(* CODESYS project e!C_CanLayer2_Test_1.ecp

Project tree, tasks and I/O mapping:
  Controller : 750-8206 PFC200 2ETH RS CAN DPS, WAGO, order no. 0750-8206, version 5.11.1.16
    application Application
      task PLC_Task (cyclic, interval t#10ms, priority 14) calls PLC_PRG
      program PLC_PRG [CFC]
      data type typCanLayer2RxSchedule
      data type typCanLayer2TxSchedule
      global variables GVL_Constants
      program CAN_Layer2_Driver [ST]: CanLayer2RxScheduler, CanLayer2TxScheduler
      global variables GVL_Variables
      data type typCanMsg
    DeviceAdapter
    Kbus : Kbus, WAGO, version 1.4.0.2
        unmapped channels: K-BUS diagnostics
      _8_DO_DI_Generic : 075x-8DO8DI, WAGO, order no. 075x-8DO8DI, version 0.0.0.13
          settings: K-BUS Module slot index = 1
          unmapped channels: _IN, _OUT
        DeviceAdapter
      RS_232_RS_485_Interface_adjustable : 0750-0652, WAGO, order no. 0750-0652, version 0.0.0.25
          settings: K-BUS Module slot index = 2
          unmapped channels: _INPUTCHANNEL, _OUTPUTCHANNEL
        DeviceAdapter
    MODBUS
      MODBUS : MODBUS, WAGO, order no. n/a, version 1.1.1.15
    PROFIBUS
      PROFIBUS : PROFIBUS, WAGO, version 1.0.0.0 (disabled)
    CANbus
      WAGO_CAN_LAYER2_DEVICE : WAGO CAN Layer2 Device, WAGO, version 3.5.4.9
    Serial
      COM1 : COM1, WAGO, version 0.0.0.19
*)

// Controller/Application/typCanLayer2RxSchedule
TYPE typCanLayer2RxSchedule :
STRUCT
	udiTimeout: UDINT := 0;
	dwId: DWORD := 16#0000_0701;(* Set MSB = TRUE if 29bit ID:  dwId = 16#8xxx_xxxx *)
	diPktCnt: DINT;
	diPktCnt_old: DINT;
	diPktDeltaCnt: DINT;
	diRegisterIdResult: CANCFG.eCanFnReturn := CanNoIdx;
	udiPktDeltaTime: UDINT; (* Delta time between each packet in one channel, in msec *)
	udiPktArrivalTime: UDINT; (* Arrival time between each packet in one channel, in msec *)
	udiPktArrivalTime_old: UDINT; (* Last arrival time between each packet in one channel, in msec *)
	TON_CanRxMonitor: TON;
	tCanRxMonitorTimeout: TIME := T#5S;
	tCanRxMonitorElapsed: TIME;
	xCanRxMonitorAlarm: BOOL;
	atypMsgFifo: ARRAY[1..GVL_Constants.LIM_OF_CANJ1939_MSG_FIFO] OF typCanMsg;
	abMsg: ARRAY [1..8] OF BYTE;
END_STRUCT
END_TYPE

// Controller/Application/typCanLayer2TxSchedule
TYPE typCanLayer2TxSchedule :
STRUCT
	TON_TxErrorMonitor : TON;
	TON_TxCyclicMonitor : TON;
	TON_TxGapMonitor : TON;
	tTxError : TIME := T#5000MS;
	tTxInterval : TIME := T#200MS;
	tTxMinGap : TIME := T#100MS;
	udiTimeout: UDINT := 0;
	bScheduleType: BYTE := 1; (* 1 = cyclic,  2 = event *)
	xTxEvent: BOOL; (* send trigger,  only valid if bScheduleType = 2 *)
	dwId: DWORD := 16#0000_0240;(* Set MSB = TRUE if 29bit ID:  dwId = 16#8xxx_xxxx *)
	dwDlc: DWORD := 3;
	diPktCnt: DINT;
	diSendResult: DINT;
	diRegisterIdResult: CANCFG.eCanFnReturn;
	abMsg: ARRAY [1..8] OF BYTE := [16#AA, 16#AA, 16#AA];
END_STRUCT
END_TYPE

// Controller/Application/typCanMsg
TYPE typCanMsg :
STRUCT
	abMsg: ARRAY [1..8] OF BYTE;
END_STRUCT
END_TYPE

// Controller/Application/GVL_Constants
VAR_GLOBAL CONSTANT
	LIM_OF_CAN_LAYER2_TX_CHANNELS: INT := 3;
	LIM_OF_CAN_LAYER2_RX_CHANNELS: INT := 3;
	LIM_OF_CANJ1939_MSG_FIFO: INT := 20;
END_VAR

// Controller/Application/GVL_Variables
VAR_GLOBAL

	bEngine_A_State: BYTE;
	bEngine_A_Ctrl: BYTE;

	TON_CanRxMonitor: TON;
	tCanRxMonitorTimeout: TIME := T#5S;
	tCanRxMonitorElapsed: TIME;
	xCanRxMonitorAlarm: BOOL;
	
	atypCanLayer2RxSchedule : ARRAY[1..LIM_OF_CAN_LAYER2_RX_CHANNELS] OF typCanLayer2RxSchedule :=
		[
			(
				udiTimeout := 0,
				dwId := 16#0000_0701,
				diRegisterIdResult := CanNoIdx
			),
			(
				udiTimeout := 0,
				dwId := 16#0000_0181,
				diRegisterIdResult := CanNoIdx
			),
			(
				udiTimeout := 0,
				dwId := 16#8CF0_0300(* MSB: activates 29bit ID *),
				diRegisterIdResult := CanNoIdx
			)
		];

	atypCanLayer2TxSchedule : ARRAY[1..LIM_OF_CAN_LAYER2_TX_CHANNELS] OF typCanLayer2TxSchedule :=
		[
			(
				bScheduleType := 1,
				udiTimeout := 0,
				tTxInterval := T#500MS,
				tTxMinGap := T#100MS,
				dwId := 16#0000_0240,
				dwDlc := 3,
				abMsg := [16#AA, 16#AA, 16#AA]
			),
			(
				bScheduleType := 1,
				udiTimeout := 0,
				tTxInterval := T#500MS,
				tTxMinGap := T#100MS,
				dwId := 16#0000_0202,
				dwDlc := 3,
				abMsg := [16#BB, 16#BB, 16#BB]
			),
			(
				bScheduleType := 1,
				udiTimeout := 0,
				tTxInterval := T#500MS,
				tTxMinGap := T#100MS,
				dwId := 16#8CD0_0300(* MSB: activates 29bit ID *),
				dwDlc := 3,
				abMsg := [16#CC, 16#CC, 16#CC]
			)
		];

END_VAR

// Controller/Application/PLC_PRG
PROGRAM PLC_PRG
VAR


END_VAR

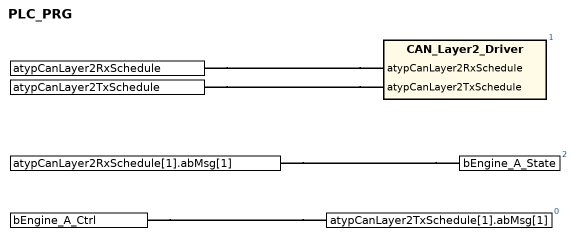
atypCanLayer2TxSchedule[1].abMsg[1] := bEngine_A_Ctrl;
CAN_Layer2_Driver(atypCanLayer2RxSchedule := atypCanLayer2RxSchedule, atypCanLayer2TxSchedule := atypCanLayer2TxSchedule);
bEngine_A_State := atypCanLayer2RxSchedule[1].abMsg[1];

END_PROGRAM

// Controller/Application/CAN_Layer2_Driver
PROGRAM CAN_Layer2_Driver
VAR_IN_OUT
	atypCanLayer2RxSchedule : ARRAY[1..LIM_OF_CAN_LAYER2_RX_CHANNELS] OF typCanLayer2RxSchedule;
	atypCanLayer2TxSchedule : ARRAY[1..LIM_OF_CAN_LAYER2_TX_CHANNELS] OF typCanLayer2TxSchedule;
END_VAR
VAR
	iCanLayer2RxChanIndex: INT;
	iCanLayer2TxChanIndex: INT;
	iCanRxPktIndex: INT;
	iCanRxPktIndexLim: INT;
	eCanL2ErrorCode: DINT;
	abMsg: ARRAY[1..8] OF BYTE;
END_VAR




CanLayer2RxScheduler();

CanLayer2TxScheduler();

ACTION CanLayer2RxScheduler:

(* Get Rx Packets *)
FOR iCanLayer2RxChanIndex := 1 TO LIM_OF_CAN_LAYER2_RX_CHANNELS DO
	IF (atypCanLayer2RxSchedule[iCanLayer2RxChanIndex].diRegisterIdResult <> CanFnOk) THEN
		(* IF CAN port is used for CAN Layer 2 and CANopen Master: *)
		(*atypCanLayer2RxSchedule[iCanLayer2RxChanIndex].diRegisterIdResult := WAGO_CANopen_Manager.RegisterId(eRegFlag := canRegisterId, dwId := atypCanLayer2RxSchedule[iCanLayer2RxChanIndex].dwId);*)

		(* IF CAN port is used for CAN Layer 2 and CANopen Slave: *)
		(*atypCanLayer2RxSchedule[iCanLayer2RxChanIndex].diRegisterIdResult := WAGO_CANopen_Local_Device.RegisterId(eRegFlag := canRegisterId, dwId := atypCanLayer2RxSchedule[iCanLayer2RxChanIndex].dwId);*)

		(* IF CAN port is used for CAN Layer 2 only: *)
		atypCanLayer2RxSchedule[iCanLayer2RxChanIndex].diRegisterIdResult := WAGO_CAN_LAYER2_Device.RegisterId(eRegFlag := canRegisterId, dwId := atypCanLayer2RxSchedule[iCanLayer2RxChanIndex].dwId);
	END_IF
	IF (atypCanLayer2RxSchedule[iCanLayer2RxChanIndex].diRegisterIdResult = CanFnOk) THEN
		GVL_Variables.TON_CanRxMonitor(IN:= TRUE, PT := GVL_Variables.tCanRxMonitorTimeout, ET=> GVL_Variables.tCanRxMonitorElapsed, Q=> GVL_Variables.xCanRxMonitorAlarm);
		atypCanLayer2RxSchedule[iCanLayer2RxChanIndex].TON_CanRxMonitor(IN:= TRUE, PT := atypCanLayer2RxSchedule[iCanLayer2RxChanIndex].tCanRxMonitorTimeout, ET=> atypCanLayer2RxSchedule[iCanLayer2RxChanIndex].tCanRxMonitorElapsed, Q=> atypCanLayer2RxSchedule[iCanLayer2RxChanIndex].xCanRxMonitorAlarm);
		(* IF CAN port is used for CAN Layer 2 and CANopen Master: *)
		(*atypCanLayer2RxSchedule[iCanLayer2RxChanIndex].diPktCnt := WAGO_CANopen_Manager.GetFrameCounter(dwId := atypCanLayer2RxSchedule[iCanLayer2RxChanIndex].dwId);*)

		(* IF CAN port is used for CAN Layer 2 and CANopen Slave: *)
		(*atypCanLayer2RxSchedule[iCanLayer2RxChanIndex].diPktCnt := WAGO_CANopen_Local_Device.GetFrameCounter(dwId := atypCanLayer2RxSchedule[iCanLayer2RxChanIndex].dwId);*)

		(* IF CAN port is used for CAN Layer 2 only: *)
		atypCanLayer2RxSchedule[iCanLayer2RxChanIndex].diPktCnt := WAGO_CAN_LAYER2_Device.GetFrameCounter(dwId := atypCanLayer2RxSchedule[iCanLayer2RxChanIndex].dwId);

		IF (atypCanLayer2RxSchedule[iCanLayer2RxChanIndex].diPktCnt <> atypCanLayer2RxSchedule[iCanLayer2RxChanIndex].diPktCnt_old) THEN
			atypCanLayer2RxSchedule[iCanLayer2RxChanIndex].TON_CanRxMonitor(IN:= FALSE);
			GVL_Variables.TON_CanRxMonitor(IN:= FALSE);
			atypCanLayer2RxSchedule[iCanLayer2RxChanIndex].diPktDeltaCnt := atypCanLayer2RxSchedule[iCanLayer2RxChanIndex].diPktCnt - atypCanLayer2RxSchedule[iCanLayer2RxChanIndex].diPktCnt_old;
			iCanRxPktIndexLim := DINT_TO_INT(MIN(MAX(0, atypCanLayer2RxSchedule[iCanLayer2RxChanIndex].diPktDeltaCnt), GVL_Constants.LIM_OF_CANJ1939_MSG_FIFO));
			FOR iCanRxPktIndex := 1 TO iCanRxPktIndexLim DO
				(* IF CAN port is used for CAN Layer 2 and CANopen Master: *)
				(*eCanL2ErrorCode := WAGO_CANopen_Manager.GetFrame(udiTimeout := atypCanLayer2RxSchedule[iCanLayer2RxChanIndex].udiTimeout, dwId := atypCanLayer2RxSchedule[iCanLayer2RxChanIndex].dwId, aMsg := abMsg);*)
	
				(* IF CAN port is used for CAN Layer 2 and CANopen Slave: *)
				(*eCanL2ErrorCode := WAGO_CANopen_Local_Device.GetFrame(udiTimeout := atypCanLayer2RxSchedule[iCanLayer2RxChanIndex].udiTimeout, dwId := atypCanLayer2RxSchedule[iCanLayer2RxChanIndex].dwId, aMsg := abMsg);*)
				
				(* IF CAN port is used for CAN Layer 2 only: *)
				eCanL2ErrorCode := WAGO_CAN_LAYER2_Device.GetFrame(udiTimeout := atypCanLayer2RxSchedule[iCanLayer2RxChanIndex].udiTimeout, dwId := atypCanLayer2RxSchedule[iCanLayer2RxChanIndex].dwId, aMsg := abMsg);

				IF ((eCanL2ErrorCode > 1) AND (eCanL2ErrorCode <= 8)) THEN
					atypCanLayer2RxSchedule[iCanLayer2RxChanIndex].abMsg := abMsg;
					atypCanLayer2RxSchedule[iCanLayer2RxChanIndex].atypMsgFifo[iCanRxPktIndex].abMsg := atypCanLayer2RxSchedule[iCanLayer2RxChanIndex].abMsg;
				END_IF
			END_FOR
			atypCanLayer2RxSchedule[iCanLayer2RxChanIndex].diPktCnt_old := atypCanLayer2RxSchedule[iCanLayer2RxChanIndex].diPktCnt;
			atypCanLayer2RxSchedule[iCanLayer2RxChanIndex].udiPktArrivalTime := TIME_TO_UDINT(TIME());
			atypCanLayer2RxSchedule[iCanLayer2RxChanIndex].udiPktDeltaTime := atypCanLayer2RxSchedule[iCanLayer2RxChanIndex].udiPktArrivalTime - atypCanLayer2RxSchedule[iCanLayer2RxChanIndex].udiPktArrivalTime_old;
			atypCanLayer2RxSchedule[iCanLayer2RxChanIndex].udiPktArrivalTime_old := atypCanLayer2RxSchedule[iCanLayer2RxChanIndex].udiPktArrivalTime;
		END_IF
	END_IF
END_FOR
END_ACTION

ACTION CanLayer2TxScheduler:


(* Send Tx Packets *)
FOR iCanLayer2TxChanIndex := 1 TO LIM_OF_CAN_LAYER2_TX_CHANNELS DO
	atypCanLayer2TxSchedule[iCanLayer2TxChanIndex].TON_TxCyclicMonitor(IN:= (atypCanLayer2TxSchedule[iCanLayer2TxChanIndex].bScheduleType = 1), PT:= atypCanLayer2TxSchedule[iCanLayer2TxChanIndex].tTxInterval);
	atypCanLayer2TxSchedule[iCanLayer2TxChanIndex].TON_TxGapMonitor(IN:= (atypCanLayer2TxSchedule[iCanLayer2TxChanIndex].bScheduleType = 2), PT:= atypCanLayer2TxSchedule[iCanLayer2TxChanIndex].tTxMinGap);
	IF ( 	(atypCanLayer2TxSchedule[iCanLayer2TxChanIndex].TON_TxCyclicMonitor.Q = TRUE) OR
			((atypCanLayer2TxSchedule[iCanLayer2TxChanIndex].xTxEvent = TRUE) AND (atypCanLayer2TxSchedule[iCanLayer2TxChanIndex].TON_TxGapMonitor.Q = TRUE))	) THEN
		atypCanLayer2TxSchedule[iCanLayer2TxChanIndex].TON_TxCyclicMonitor(IN:= FALSE);
		IF (atypCanLayer2TxSchedule[iCanLayer2TxChanIndex].xTxEvent = TRUE) THEN
			atypCanLayer2TxSchedule[iCanLayer2TxChanIndex].xTxEvent := FALSE;
			atypCanLayer2TxSchedule[iCanLayer2TxChanIndex].TON_TxGapMonitor(IN:= FALSE);
		END_IF

		(* IF CAN port is used for CAN Layer 2 and CANopen Master: *)
		(*atypCanLayer2TxSchedule[iCanLayer2TxChanIndex].diSendResult := WAGO_CANopen_Manager.SendFrame(dwId := atypCanLayer2TxSchedule[iCanLayer2TxChanIndex].dwId, dwDlc := atypCanLayer2TxSchedule[iCanLayer2TxChanIndex].dwDlc, udiTimeout := atypCanLayer2TxSchedule[iCanLayer2TxChanIndex].udiTimeout, aMsg := atypCanLayer2TxSchedule[iCanLayer2TxChanIndex].abMsg);*)

		(* IF CAN port is used for CAN Layer 2 and CANopen Slave: *)
		(*atypCanLayer2TxSchedule[iCanLayer2TxChanIndex].diSendResult := WAGO_CANopen_Local_Device.SendFrame(dwId := atypCanLayer2TxSchedule[iCanLayer2TxChanIndex].dwId, dwDlc := atypCanLayer2TxSchedule[iCanLayer2TxChanIndex].dwDlc, udiTimeout := atypCanLayer2TxSchedule[iCanLayer2TxChanIndex].udiTimeout, aMsg := atypCanLayer2TxSchedule[iCanLayer2TxChanIndex].abMsg);*)

		(* IF CAN port is used for CAN Layer 2 only: *)
		atypCanLayer2TxSchedule[iCanLayer2TxChanIndex].diSendResult := WAGO_CAN_LAYER2_Device.SendFrame(dwId := atypCanLayer2TxSchedule[iCanLayer2TxChanIndex].dwId, dwDlc := atypCanLayer2TxSchedule[iCanLayer2TxChanIndex].dwDlc, udiTimeout := atypCanLayer2TxSchedule[iCanLayer2TxChanIndex].udiTimeout, aMsg := atypCanLayer2TxSchedule[iCanLayer2TxChanIndex].abMsg);

		atypCanLayer2TxSchedule[iCanLayer2TxChanIndex].diPktCnt := atypCanLayer2TxSchedule[iCanLayer2TxChanIndex].diPktCnt + 1;
		iCanLayer2TxChanIndex := iCanLayer2TxChanIndex + 1;
	END_IF
END_FOR
END_ACTION

END_PROGRAM
